PROGRAM MAIN
VAR
END_VAR

END_PROGRAM

(* stored: Version 1.1.0.1, ProductVersion 3.1.4024.12
   POU MAIN: Id {d4df455a-6e4a-477c-86c3-a104380c461f}, SpecialFunc None *)
